FUNCTION_BLOCK SORTER_GET_COLOR (* Basic Function Block Type *)
  (* Standard: 61499-2 *)
  (* Version 0.0, 1/17/2023, brink, Flexbridge AB, Template *)
  PACKAGE UAO.Hackathon;
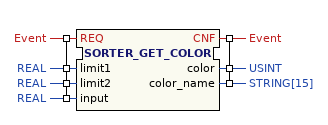
  EVENT_INPUT
    REQ WITH limit1, limit2, input; (* Normal Execution Request *)
  END_EVENT
  EVENT_OUTPUT
    CNF WITH color, color_name; (* Execution Confirmation *)
  END_EVENT
  VAR_INPUT
    limit1 : REAL;
    limit2 : REAL;
    input : REAL; (* Input value from analog sensor *)
  END_VAR
  VAR_OUTPUT
    color : USINT;
    color_name : STRING[15];
  END_VAR
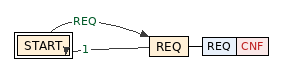
  EC_STATES
    START; (* Initial State *)
    REQ : REQ -> CNF; (* Normal execution *)
  END_STATES
  EC_TRANSITIONS
    START TO REQ := REQ;
    REQ TO START := 1;
  END_TRANSITIONS
  ALGORITHM REQ IN ST: (* Normally executed algorithm *)
IF input <= limit1 THEN
    color := 0;
    color_name :='white';
ELSIF input <= limit2 THEN
	color := 1;
    color_name :='red';
ELSE
	color := 2;
    color_name :='blue';
END_IF;
  END_ALGORITHM
END_FUNCTION_BLOCK
